# EPICS IOC start-up script: examples/test/PSI/ep3162.iocsh
#- mXsXXX naming
require ecmccfg v7_RC1, "NAMING=mXsXXX"

#- add slaves
${SCRIPTEXEC} ${ecmccfg_DIR}addSlave.cmd, "HW_DESC=EP3162, SLAVE_ID=${SLAVE=0}"
